// SIMATIC S7-200 SMART project (STEP 7-Micro/WIN SMART), CPU ST60

SYMBOL_TABLE 系统符号
Always_On        SM0.0    // 始终接通
First_Scan_On    SM0.1    // 仅在第一个扫描周期时接通
END_SYMBOL_TABLE

ORGANIZATION_BLOCK MAIN:OB1
TITLE=程序注释
BEGIN
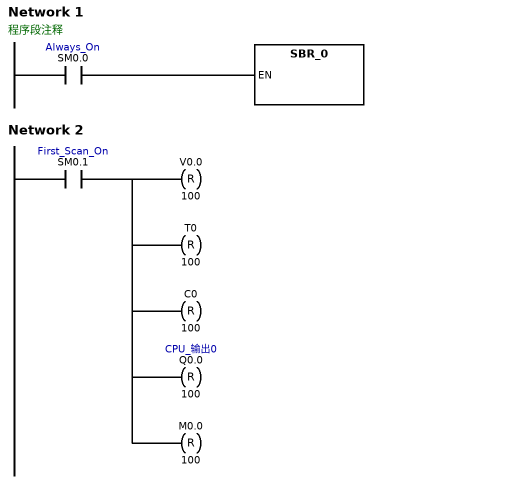
Network 1
// 程序段注释
LD     Always_On:SM0.0
CALL   SBR_0:SBR0
Network 2
LD     First_Scan_On:SM0.1
R      V0.0, 100
R      T0, 100
R      C0, 100
R      CPU_输出0:Q0.0, 100
R      M0.0, 100
END_ORGANIZATION_BLOCK

SUBROUTINE_BLOCK SBR_0:SBR0
TITLE=子程序注释
BEGIN
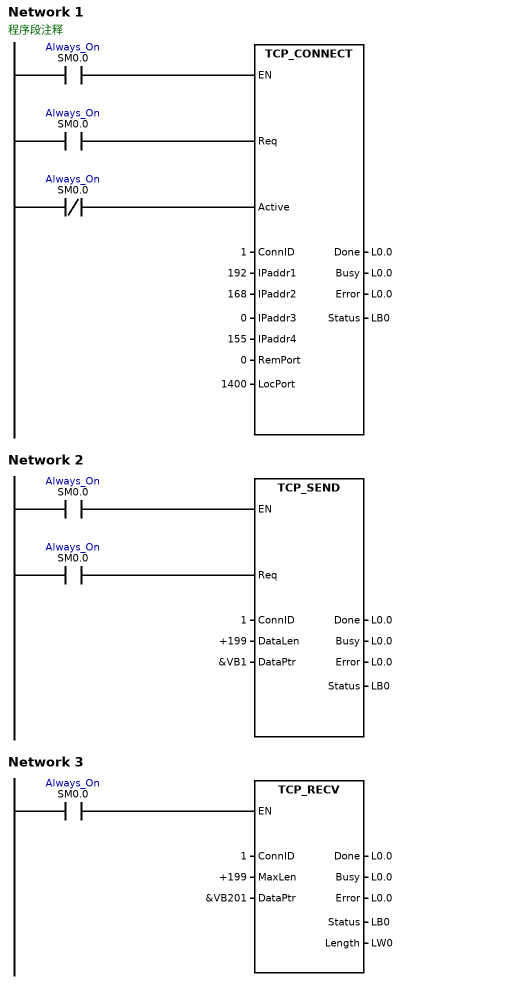
Network 1
// 程序段注释
LD     Always_On:SM0.0
=      L60.0
LD     Always_On:SM0.0
=      L63.7
LDN    Always_On:SM0.0
=      L63.6
LD     L60.0
CALL   TCP_CONNECT:SBR4, L63.7, L63.6, 1, 192, 168, 0, 155, 0, 1400, L0.0, L0.0, L0.0, LB0
Network 2
LD     Always_On:SM0.0
=      L60.0
LD     Always_On:SM0.0
=      L63.7
LD     L60.0
CALL   TCP_SEND:SBR5, L63.7, 1, +199, &VB1, L0.0, L0.0, L0.0, LB0
Network 3
LD     Always_On:SM0.0
CALL   TCP_RECV:SBR6, 1, +199, &VB201, L0.0, L0.0, L0.0, LB0, LW0
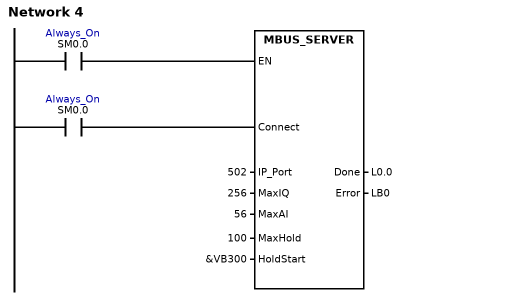
Network 4
LD     Always_On:SM0.0
=      L60.0
LD     Always_On:SM0.0
=      L63.7
LD     L60.0
CALL   MBUS_SERVER:SBR8, L63.7, 502, 256, 56, 100, &VB300, L0.0, LB0
END_SUBROUTINE_BLOCK

SUBROUTINE_BLOCK SBR_1:SBR1
TITLE=子程序注释
BEGIN
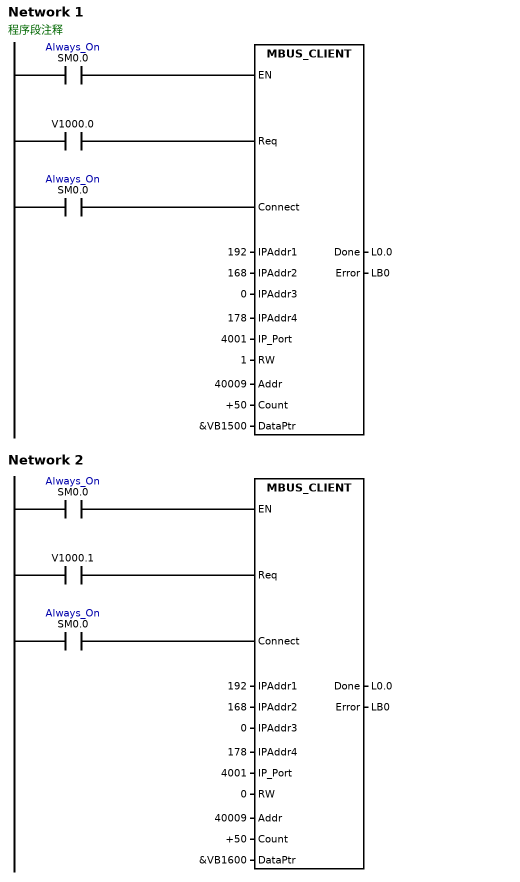
Network 1
// 程序段注释
LD     Always_On:SM0.0
=      L60.0
LD     V1000.0
=      L63.7
LD     Always_On:SM0.0
=      L63.6
LD     L60.0
CALL   MBUS_CLIENT:SBR7, L63.7, L63.6, 192, 168, 0, 178, 4001, 1, 40009, +50, &VB1500, L0.0, LB0
Network 2
LD     Always_On:SM0.0
=      L60.0
LD     V1000.1
=      L63.7
LD     Always_On:SM0.0
=      L63.6
LD     L60.0
CALL   MBUS_CLIENT:SBR7, L63.7, L63.6, 192, 168, 0, 178, 4001, 0, 40009, +50, &VB1600, L0.0, LB0
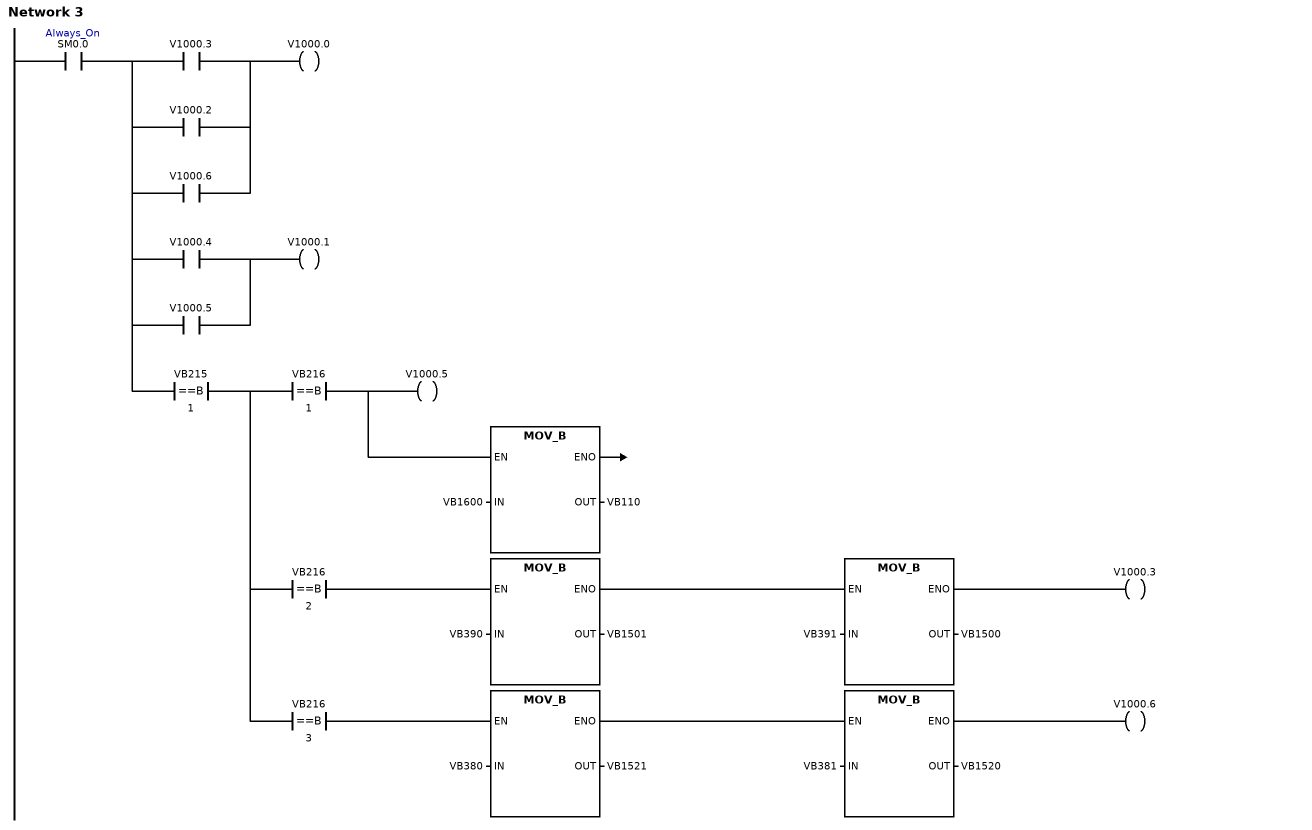
Network 3
LD     Always_On:SM0.0
LPS
LD     V1000.3
O      V1000.2
O      V1000.6
ALD
=      V1000.0
LRD
LD     V1000.4
O      V1000.5
ALD
=      V1000.1
LPP
AB=    VB215, 1
LPS
AB=    VB216, 1
=      V1000.5
MOVB   VB1600, VB110
LPP
LPS
AB=    VB216, 2
MOVB   VB390, VB1501
AENO
MOVB   VB391, VB1500
AENO
=      V1000.3
LPP
AB=    VB216, 3
MOVB   VB380, VB1521
AENO
MOVB   VB381, VB1520
AENO
=      V1000.6
END_SUBROUTINE_BLOCK

SUBROUTINE_BLOCK SBR_2:SBR2
TITLE=子程序注释
BEGIN
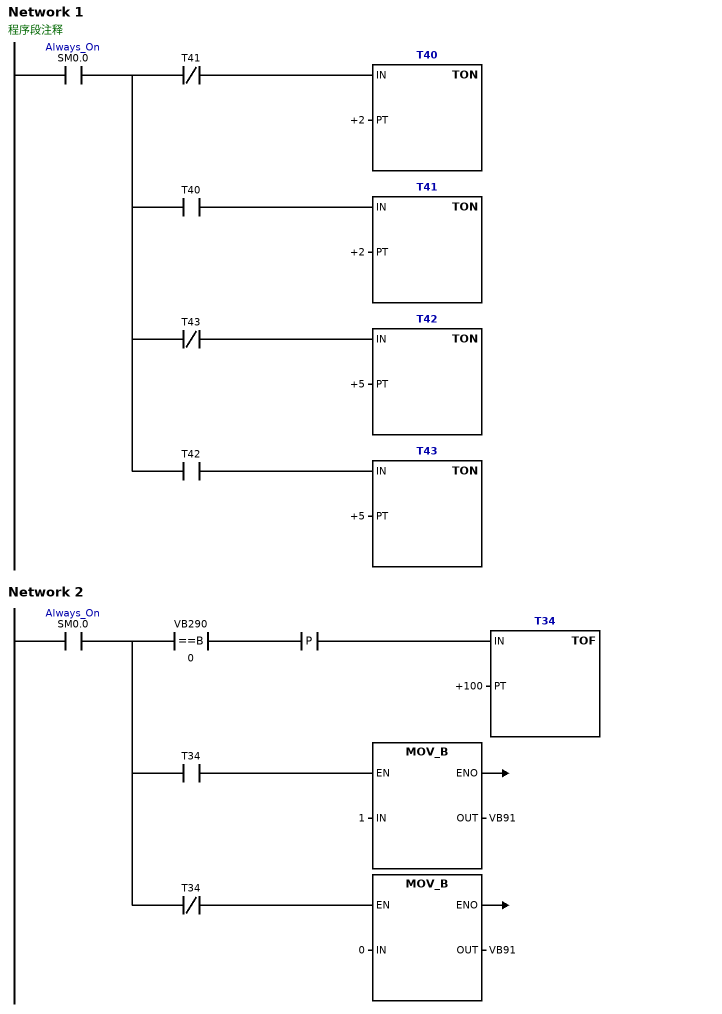
Network 1
// 程序段注释
LD     Always_On:SM0.0
LPS
AN     T41
TON    T40, +2
LRD
A      T40
TON    T41, +2
LRD
AN     T43
TON    T42, +5
LPP
A      T42
TON    T43, +5
Network 2
LD     Always_On:SM0.0
LPS
AB=    VB290, 0
EU
TOF    T34, +100
LRD
A      T34
MOVB   1, VB91
LPP
AN     T34
MOVB   0, VB91
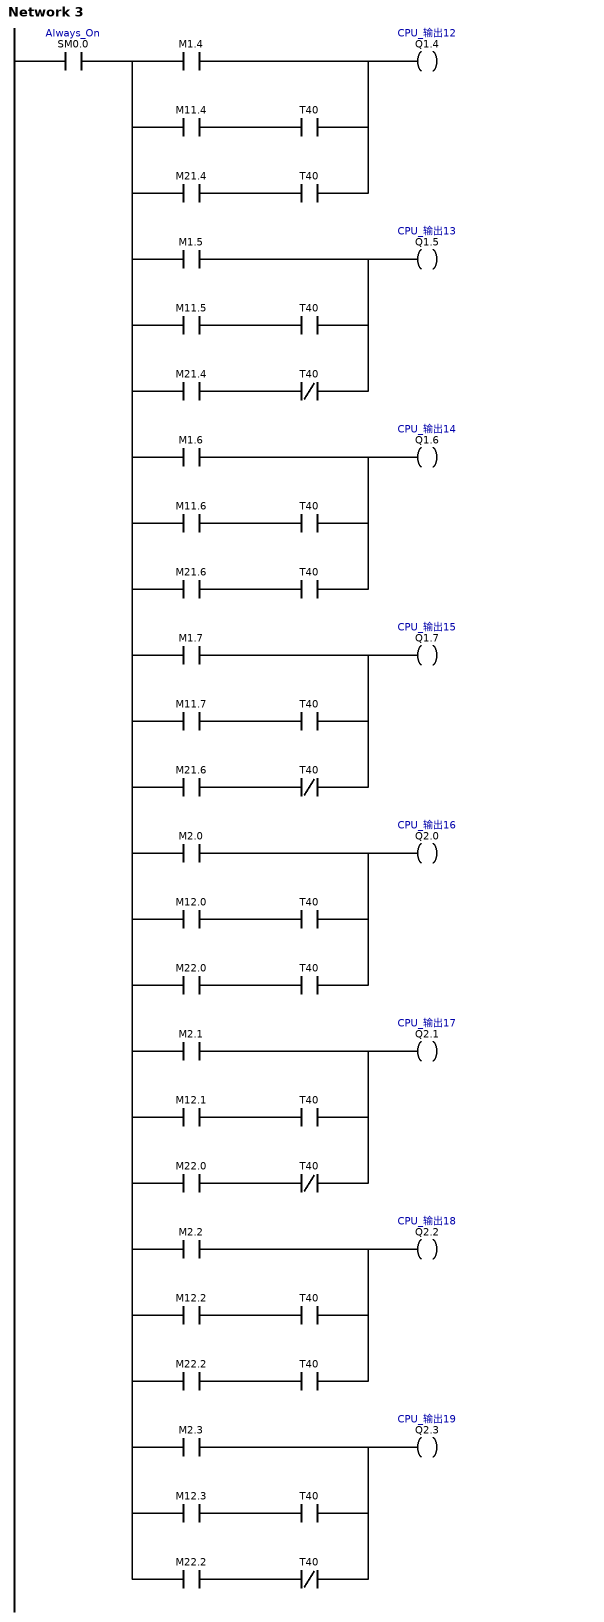
Network 3
LD     Always_On:SM0.0
LPS
LD     M1.4
LD     M11.4
A      T40
OLD
LD     M21.4
A      T40
OLD
ALD
=      CPU_输出12:Q1.4
LRD
LD     M1.5
LD     M11.5
A      T40
OLD
LD     M21.4
AN     T40
OLD
ALD
=      CPU_输出13:Q1.5
LRD
LD     M1.6
LD     M11.6
A      T40
OLD
LD     M21.6
A      T40
OLD
ALD
=      CPU_输出14:Q1.6
LRD
LD     M1.7
LD     M11.7
A      T40
OLD
LD     M21.6
AN     T40
OLD
ALD
=      CPU_输出15:Q1.7
LRD
LD     M2.0
LD     M12.0
A      T40
OLD
LD     M22.0
A      T40
OLD
ALD
=      CPU_输出16:Q2.0
LRD
LD     M2.1
LD     M12.1
A      T40
OLD
LD     M22.0
AN     T40
OLD
ALD
=      CPU_输出17:Q2.1
LRD
LD     M2.2
LD     M12.2
A      T40
OLD
LD     M22.2
A      T40
OLD
ALD
=      CPU_输出18:Q2.2
LPP
LD     M2.3
LD     M12.3
A      T40
OLD
LD     M22.2
AN     T40
OLD
ALD
=      CPU_输出19:Q2.3
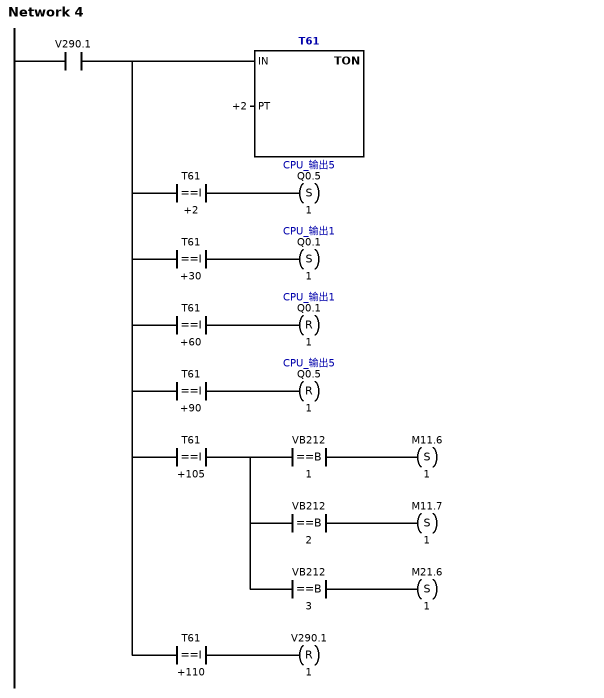
Network 4
LD     V290.1
LPS
TON    T61, +2
AW=    T61, +2
S      CPU_输出5:Q0.5, 1
LRD
AW=    T61, +30
S      CPU_输出1:Q0.1, 1
LRD
AW=    T61, +60
R      CPU_输出1:Q0.1, 1
LRD
AW=    T61, +90
R      CPU_输出5:Q0.5, 1
LRD
AW=    T61, +105
LPS
AB=    VB212, 1
S      M11.6, 1
LRD
AB=    VB212, 2
S      M11.7, 1
LPP
AB=    VB212, 3
S      M21.6, 1
LPP
AW=    T61, +110
R      V290.1, 1
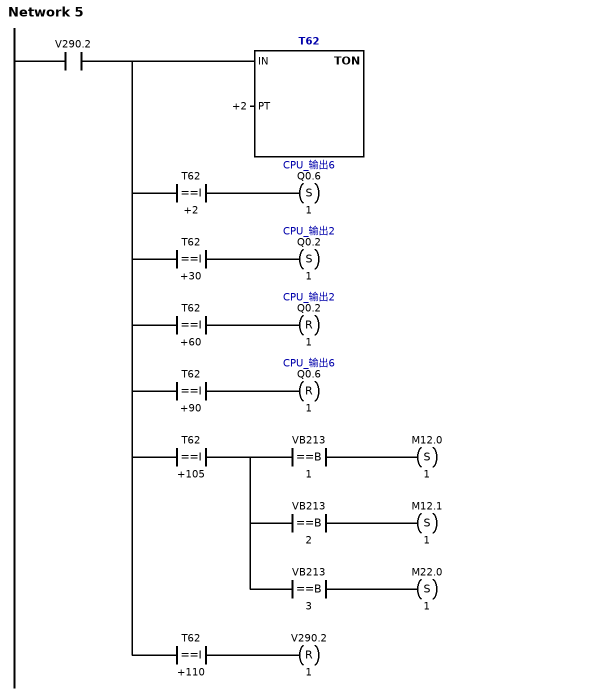
Network 5
LD     V290.2
LPS
TON    T62, +2
AW=    T62, +2
S      CPU_输出6:Q0.6, 1
LRD
AW=    T62, +30
S      CPU_输出2:Q0.2, 1
LRD
AW=    T62, +60
R      CPU_输出2:Q0.2, 1
LRD
AW=    T62, +90
R      CPU_输出6:Q0.6, 1
LRD
AW=    T62, +105
LPS
AB=    VB213, 1
S      M12.0, 1
LRD
AB=    VB213, 2
S      M12.1, 1
LPP
AB=    VB213, 3
S      M22.0, 1
LPP
AW=    T62, +110
R      V290.2, 1
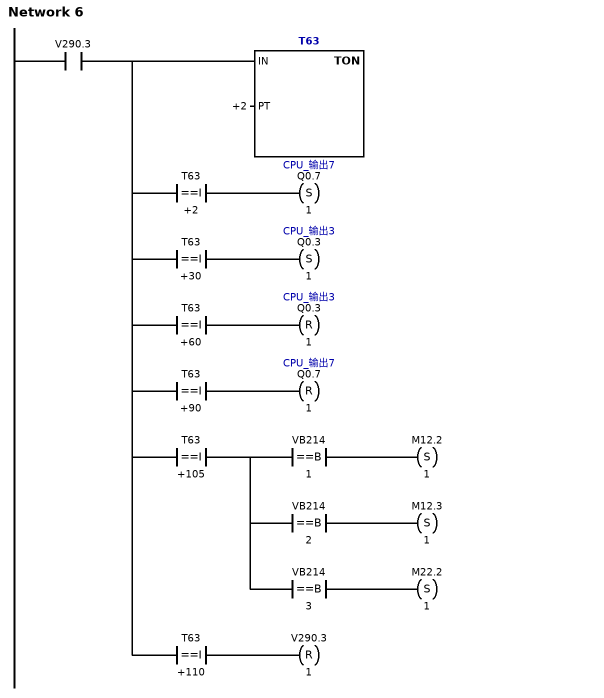
Network 6
LD     V290.3
LPS
TON    T63, +2
AW=    T63, +2
S      CPU_输出7:Q0.7, 1
LRD
AW=    T63, +30
S      CPU_输出3:Q0.3, 1
LRD
AW=    T63, +60
R      CPU_输出3:Q0.3, 1
LRD
AW=    T63, +90
R      CPU_输出7:Q0.7, 1
LRD
AW=    T63, +105
LPS
AB=    VB214, 1
S      M12.2, 1
LRD
AB=    VB214, 2
S      M12.3, 1
LPP
AB=    VB214, 3
S      M22.2, 1
LPP
AW=    T63, +110
R      V290.3, 1
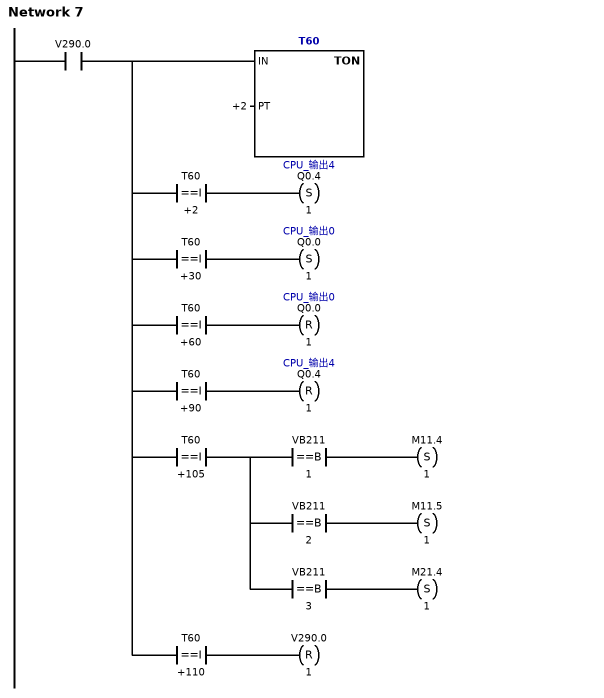
Network 7
LD     V290.0
LPS
TON    T60, +2
AW=    T60, +2
S      CPU_输出4:Q0.4, 1
LRD
AW=    T60, +30
S      CPU_输出0:Q0.0, 1
LRD
AW=    T60, +60
R      CPU_输出0:Q0.0, 1
LRD
AW=    T60, +90
R      CPU_输出4:Q0.4, 1
LRD
AW=    T60, +105
LPS
AB=    VB211, 1
S      M11.4, 1
LRD
AB=    VB211, 2
S      M11.5, 1
LPP
AB=    VB211, 3
S      M21.4, 1
LPP
AW=    T60, +110
R      V290.0, 1
END_SUBROUTINE_BLOCK

SUBROUTINE_BLOCK SBR_3:SBR3
TITLE=子程序注释
BEGIN
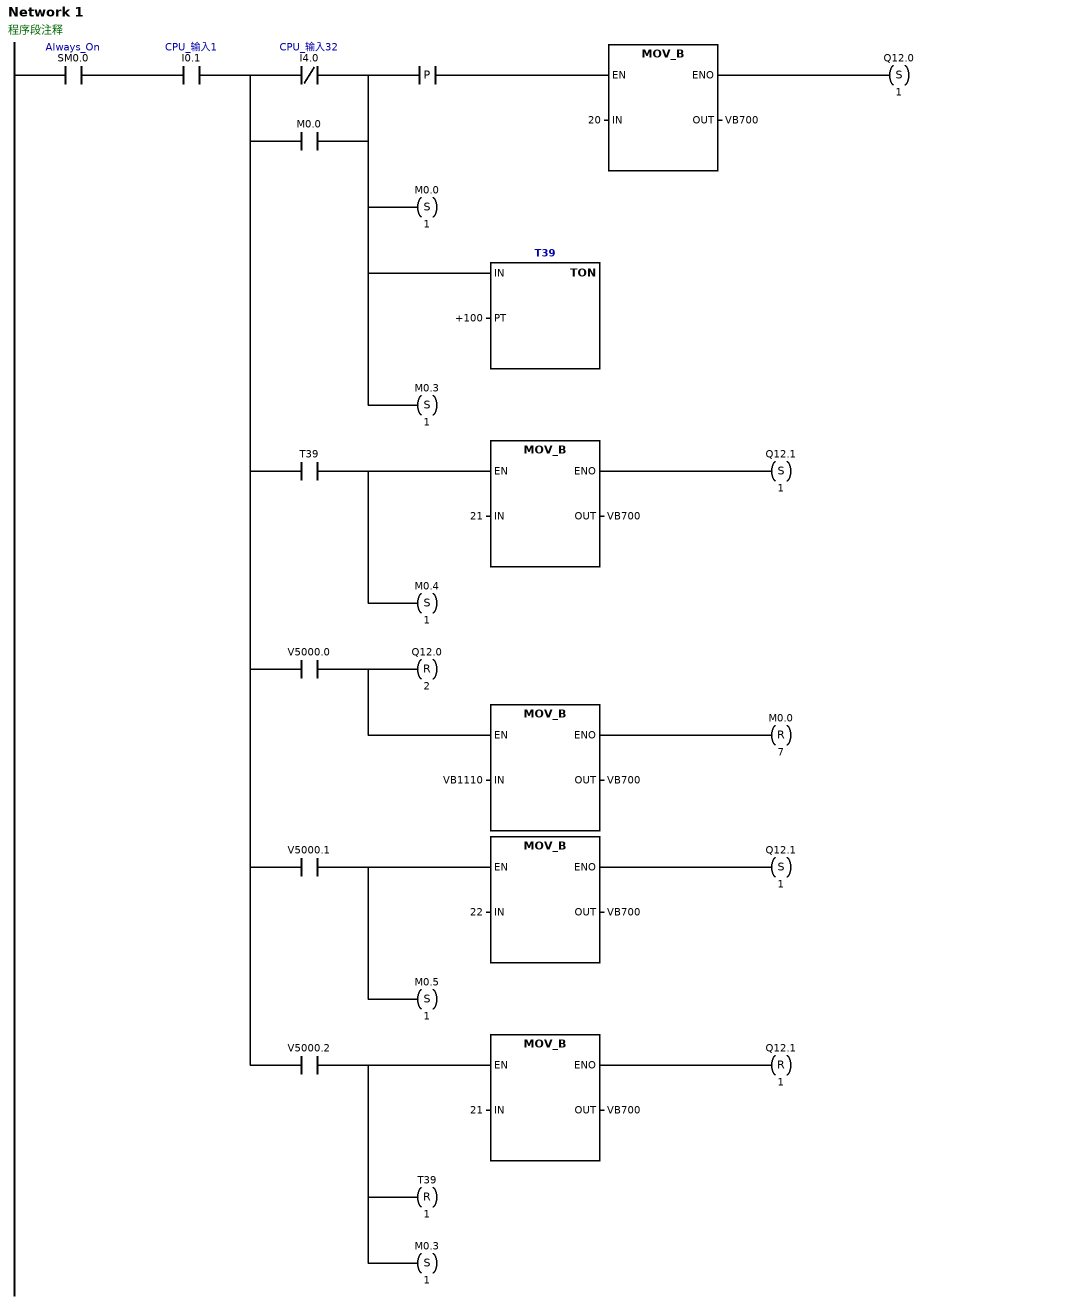
Network 1
// 程序段注释
LD     Always_On:SM0.0
A      CPU_输入1:I0.1
LPS
LDN    CPU_输入32:I4.0
O      M0.0
ALD
LPS
EU
MOVB   20, VB700
AENO
S      Q12.0, 1
LRD
S      M0.0, 1
LRD
TON    T39, +100
LPP
S      M0.3, 1
LRD
A      T39
LPS
MOVB   21, VB700
AENO
S      Q12.1, 1
LPP
S      M0.4, 1
LRD
A      V5000.0
R      Q12.0, 2
MOVB   VB1110, VB700
AENO
R      M0.0, 7
LRD
A      V5000.1
LPS
MOVB   22, VB700
AENO
S      Q12.1, 1
LPP
S      M0.5, 1
LPP
A      V5000.2
LPS
MOVB   21, VB700
AENO
R      Q12.1, 1
LRD
R      T39, 1
LPP
S      M0.3, 1
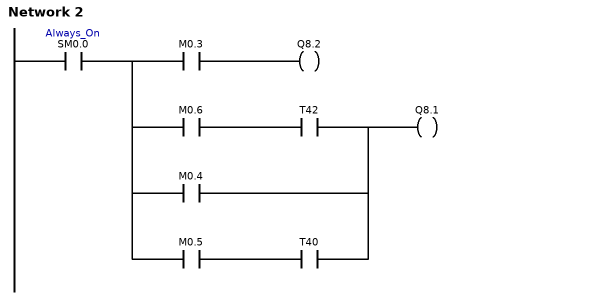
Network 2
LD     Always_On:SM0.0
LPS
A      M0.3
=      Q8.2
LPP
LD     M0.6
A      T42
O      M0.4
LD     M0.5
A      T40
OLD
ALD
=      Q8.1
END_SUBROUTINE_BLOCK

// SBR4: protected block, not included

// SBR5: protected block, not included

// SBR6: protected block, not included

// SBR7: protected block, not included

// SBR8: protected block, not included
